// TIA Portal V20 export
DATA_BLOCK "DB_NordSetPoint"   // DB34
// stored: Access Published, MemoryReserve 100, Namespace LineC1
   VAR
      Line : Struct
         C1 : Struct   // -(0 - 16000) -> (CW: 0 - 100%) || +(0 - 16000) (CCW: 0 - 100%) || freq. has been set via NORDCON
            Conveyor : Array[_.minC1.._.maxC1] of DInt;
         END_STRUCT;
      END_STRUCT;
   END_VAR
BEGIN
END_DATA_BLOCK
